FUNCTION FrameIsValid : BOOL
VAR_INPUT
	frame : REFERENCE TO VisionFrame;
END_VAR
VAR
	emptyFrame : VisionFrame;
END_VAR

FrameIsValid := 
	MEMCMP(ADR(frame), ADR(emptyFrame), SIZEOF(VisionFrame)) <> 0 OR
	frame.MaterialID = '' OR
	frame.CheckFor = '' OR
	frame.CameraNumber = 0;

END_FUNCTION

(* stored: Version 1.1.0.1, ProductVersion 3.1.4024.11
   POU FrameIsValid: Id {7ffde625-7111-4b70-aa34-bd80f0f00da2}, SpecialFunc None *)
